// TwinCAT 3 PLC project log4Tc_Tester
// ProgramVersion: 3.1.4026.12
// CompilerDefines: DEBUG
// libraries:
//   Tc2_Standard, * (Beckhoff Automation GmbH)
//   Tc2_System, * (Beckhoff Automation GmbH)
//   Tc2_Utilities, * (Beckhoff Automation GmbH)
//   Tc3_Module, * (Beckhoff Automation GmbH)
//   [log4TC], * (mbc engineering)
//   Base Interfaces,newest,System
// project tree:
//   GVLs/ GVL.TcGVL
//   / PlcTask.TcTTO
//   POUs/ CheckBounds.TcPOU, CheckLRangeSigned.TcPOU, CheckLRangeUnsigned.TcPOU, CheckPointer.TcPOU, CheckRangeSigned.TcPOU, CheckRangeUnsigned.TcPOU, FB_TcExternalTime.TcPOU, F_FUN.TcPOU, MAIN.TcPOU, PRG_TestSimpleApi.TcPOU
// (motion and I/O tree: see PLC project mbc_log4tc)
// real-time tasks:
//   TASK PlcTask: cycle T#1ms, priority 20, ADS port 350
//   TASK PlcTask1: cycle T#10ms, priority 21, ADS port 351

CONFIGURATION log4Tc_Tester
    RESOURCE PLC ON TwinCAT3
        TASK PlcTask(INTERVAL := T#1ms, PRIORITY := 20);
        PROGRAM MAIN WITH PlcTask : MAIN;
    END_RESOURCE
END_CONFIGURATION

// ---- GVLs/GVL.TcGVL
{attribute 'qualified_only'}
VAR_GLOBAL
END_VAR

// ---- POUs/MAIN.TcPOU
PROGRAM MAIN
VAR
	fbTime			: FB_TcExternalTime(ETcExternalTimeType.SystemTime);
	nOffset			: LINT;
	bWriteLog		: BOOL;
	bWriteCont		: BOOL;
	nVar1			: INT;
	nVar2			: T_MaxString := 'ä';
	nVar3			: REAL;
	var1			: __SYSTEM.VAR_INFO;
	b1 : BYTE;
	b2 : BYTE;
END_VAR

IF _TaskInfo[GETCURTASKINDEXEX()].FirstCycle THEN
	// For Remote Log4TC Server change the AMS net ID and configure a route
	// PRG_TaskLog.Init('127.0.0.1.1.1');
	F_Log(E_LogLevel.eInfo, 'Started');
END_IF


PRG_TestSimpleApi();
	

PRG_TaskLog.Call();

END_PROGRAM

// ---- POUs/FB_TcExternalTime.TcPOU
FUNCTION_BLOCK FB_TcExternalTime
VAR
	_hr : HRESULT;
	_ipExtTime : ITcExternalTime;
	_eTimeType: ETcExternalTimeType;
END_VAR

METHOD FB_Exit : BOOL
VAR_INPUT
	bInCopyCode : BOOL; // if TRUE, the exit method is called for exiting an instance that is copied afterwards (online change).
END_VAR
IF _ipExtTime <> 0 THEN
	FW_SafeRelease(ADR(_ipExtTime));
END_IF
END_METHOD

METHOD FB_Init : BOOL
VAR_INPUT
	bInitRetains : BOOL; // if TRUE, the retain variables are initialized (warm start / cold start)
	bInCopyCode : BOOL;  // if TRUE, the instance afterwards gets moved into the copy code (online change)
	eTimeType : ETcExternalTimeType; 
END_VAR
VAR
	ipServer : ITComObjectServer;
END_VAR
ipServer := TwinCAT_SystemInfoVarList._AppInfo.TComSrvPtr;
_eTimeType := eTimeType; 
IF _ipExtTime = 0 THEN
	_hr := ipServer.TcQueryInterface(IID_ITcExternalTime, ADR(_ipExtTime));
	IF FAILED(_hr) THEN RETURN; END_IF
END_IF
END_METHOD

METHOD GetExternalOffset : LINT
VAR_INPUT
END_VAR
IF _ipExtTime <> 0 THEN
	_hr := _ipExtTime.GetExternalTimeOffset(_eTimeType, GetExternalOffset);
	IF _hr <> 0 THEN GetExternalOffset := 0; END_IF
END_IF
END_METHOD

METHOD GetExternalTime : LINT
VAR_INPUT
END_VAR
IF _ipExtTime <> 0 THEN
	GetExternalTime := GetSystemTime();
	_hr := _ipExtTime.SystemTimeToExternalTime(_eTimeType, GetExternalTime);
	IF _hr <> 0 THEN GetExternalTime := 0; END_IF
END_IF
END_METHOD

METHOD GetSystemTime : LINT
GetSystemTime := ULINT_TO_LINT(F_GetSystemTime());
END_METHOD

PROPERTY Result : HRESULT
GET
Result := _hr;
END_GET
END_PROPERTY

END_FUNCTION_BLOCK

// ---- POUs/PRG_TestSimpleApi.TcPOU
PROGRAM PRG_TestSimpleApi
VAR
	bExecute		: BOOL;
	bExecuteSingle	: BOOL;
	
	nArg			: INT := 42;
	sArg			: T_MaxString := 'foo';
	fArg			: REAL := 4.2;
	
	tTime			: TIME :=  T#12H34M15S;
	tLTime			: LTIME := LTIME#1000D15H23M12S34MS2US44NS;
	dDate			: DATE := DATE#1996-05-06;
	dDT				: DT := DATE_AND_TIME#1996-05-06-15:36:30;
	tTOD			: TOD := TIME_OF_DAY#15:36:30.123;
	eEnum			: E_LogLevel := E_LogLevel.eFatal;
	wStr			: WSTRING := "fooöäaΘ𝄞";
	
	fbScope			: FB_ScopedContext;
END_VAR

//fbScope.ContextBuilder.AddInt('scope', 42);

IF bExecute OR bExecuteSingle THEN
	bExecuteSingle := FALSE;

	F_LogLA1C(
		E_LogLevel.eInfo, 
		'PRG_TestSimpleApi', 
		'Temperatur {temperature}', 
		fArg, 
		F_LogContext().AddBool('csv', TRUE)
	);
	
	
	F_LogA7(
		E_LogLevel.eInfo, 
		'Neue Datentypen TIME={time} LTIME={ltime} DATE={date} DT={date_and_time} TOD={time_of_day} ENUM={enum} WSTRING={wstring}',
		tTime,
		tLTime,
		dDate,
		dDT,
		tTOD,
		eEnum,
		wStr
	);
		
		
	
	(*
	
	fbScope.Begin();
	
	F_LogLA3(
		E_LogLevel.eInfo,
		'PRG_TestSimpleApi',
		'Log F_LogLA3({arg1},{arg2},{arg3})',
		nArg,
		sArg,
		fArg,
	);
	
	fbScope.End();
	
	F_LogA3(
		E_LogLevel.eInfo,
		'Log F_LogA3({arg1},{arg2},{arg3})',
		nArg,
		sArg,
		fArg
	);
	¨*)
	
END_IF

END_PROGRAM

// ---- POUs/CheckBounds.TcPOU
// Implicitly generated code : DO NOT EDIT
FUNCTION CheckBounds : DINT
VAR_INPUT
	index, lower, upper: DINT;
END_VAR

{noflow}
IF (index < lower) THEN
	CheckBounds := lower;
	F_LogLA3(E_LogLevel.eFatal, 'CheckBounds', 'Check bounds exception: {index} {lower} {upper}', index, lower, upper);
ELSIF(index > upper) THEN
	CheckBounds := upper;
	F_LogLA3(E_LogLevel.eFatal, 'CheckBounds', 'Check bounds exception: {index} {lower} {upper}', index, lower, upper);
ELSE
	CheckBounds := index;
END_IF
{flow}

END_FUNCTION

// ---- POUs/CheckLRangeSigned.TcPOU
// Implicitly generated code : DO NOT EDIT
FUNCTION CheckLRangeSigned : LINT
VAR_INPUT
	value, lower, upper: LINT;
END_VAR

{noflow}
IF (value < lower) THEN
	CheckLRangeSigned := lower;
	F_LogLA3(E_LogLevel.eFatal, 'CheckLRangeSigned', 'Check LINT range signed exception: {value} {lower} {upper}', value, lower, upper);
ELSIF(value > upper) THEN
	CheckLRangeSigned := upper;
	F_LogLA3(E_LogLevel.eFatal, 'CheckLRangeSigned', 'Check LINT range signed exception: {value} {lower} {upper}', value, lower, upper);
ELSE
	CheckLRangeSigned := value;
END_IF
{flow}

END_FUNCTION

// ---- POUs/CheckLRangeUnsigned.TcPOU
// Implicitly generated code : DO NOT EDIT
FUNCTION CheckLRangeUnsigned : ULINT
VAR_INPUT
	value, lower, upper: ULINT;
END_VAR

{noflow}
IF (value < lower) THEN
	CheckLRangeUnsigned := lower;
	F_LogLA3(E_LogLevel.eFatal, 'CheckLRangeUnsigned', 'Check ULINT range unsigned exception: {value} {lower} {upper}', value, lower, upper);
ELSIF(value > upper) THEN
	CheckLRangeUnsigned := upper;
	F_LogLA3(E_LogLevel.eFatal, 'CheckLRangeUnsigned', 'Check ULINT range unsigned exception: {value} {lower} {upper}', value, lower, upper);
ELSE
	CheckLRangeUnsigned := value;
END_IF
{flow}

END_FUNCTION

// ---- POUs/CheckPointer.TcPOU
// Implicitly generated code : DO NOT EDIT
FUNCTION CheckPointer : POINTER TO BYTE
VAR_INPUT 
	ptToTest : POINTER TO BYTE; // Destination address of the pointer
	iSize : DINT;		        // Size of the type the pointer points to. (e.g: 20 for POINTER TO ARRAY [0..9] OF INT) 
	iGran : DINT;		        // Granularity of the pointer access. This is the size of the biggest non-structured data type in the type the pointer points to. (e.g: 2 for POINTER TO ARRAY [0..9] OF INT)
	bWrite: BOOL;		        // Indicates read or write Access. TRUE = write access.
END_VAR

IF ptToTest = 0 THEN
	F_LogLA3(E_LogLevel.eFatal, 'CheckPointer', 'Check pointer exception: {iSize} {iGran} {bWrite}', iSize, iGran, bWrite);
END_IF
CheckPointer := ptToTest;

END_FUNCTION

// ---- POUs/CheckRangeSigned.TcPOU
// Implicitly generated code : DO NOT EDIT
FUNCTION CheckRangeSigned : DINT
VAR_INPUT
	value, lower, upper: DINT;
END_VAR

{noflow}
IF (value < lower) THEN
	CheckRangeSigned := lower;
	F_LogLA3(E_LogLevel.eFatal, 'CheckRangeSigned', 'Check DINT range signed exception: {value} {lower} {upper}', value, lower, upper);
ELSIF(value > upper) THEN
	CheckRangeSigned := upper;
	F_LogLA3(E_LogLevel.eFatal, 'CheckRangeSigned', 'Check DINT range signed exception: {value} {lower} {upper}', value, lower, upper);
ELSE
	CheckRangeSigned := value;
END_IF
{flow}

END_FUNCTION

// ---- POUs/CheckRangeUnsigned.TcPOU
// Implicitly generated code : DO NOT EDIT
FUNCTION CheckRangeUnsigned : UDINT
VAR_INPUT
	value, lower, upper: UDINT;
END_VAR

{noflow}
IF (value < lower) THEN
	CheckRangeUnsigned := lower;
	F_LogLA3(E_LogLevel.eFatal, 'CheckRangeUnsigned', 'Check UDINT range unsigned exception: {value} {lower} {upper}', value, lower, upper);
ELSIF(value > upper) THEN
	CheckRangeUnsigned := upper;
	F_LogLA3(E_LogLevel.eFatal, 'CheckRangeUnsigned', 'Check UDINT range unsigned exception: {value} {lower} {upper}', value, lower, upper);
ELSE
	CheckRangeUnsigned := value;
END_IF
{flow}

END_FUNCTION

// ---- POUs/F_FUN.TcPOU
FUNCTION F_FUN : BOOL
VAR_INPUT
END_VAR
VAR
	var1			: __SYSTEM.VAR_INFO;
	var2			: __SYSTEM.VAR_INFO;
	fbLog			: FB_Logger('F_FUN (Inst)');
END_VAR
VAR_STAT
	fbLog2			: FB_Logger('F_FUN (Stat)');
END_VAR

fbLog();
fbLog2();
var1 := __VARINFO(fbLog);
var2 := __VARINFO(fbLog2);

END_FUNCTION
